(* CODESYS project SampleProject_IoDrvMasterTemplateIEC.project

Project tree, tasks and I/O mapping:
  Device : CODESYS Control Win V3, 3S - Smart Software Solutions GmbH, version 3.5.14.10
    application Application
      libraries: Standard, * (System); CAA Device Diagnosis, 3.5.15.0 (CAA Technical Workgroup)
      task MainTask (cyclic, interval t#20ms, priority 1) calls PLC_PRG
      program PLC_PRG [ST]
    My_card_IEC_Driver_master_ : My card IEC Driver (master), My company, order no. 0815, version 3.5.15.0
      Slave_without_modules_internal_8xDI_8xDO_T3 : Slave without modules (internal: 8xDI, 8xDO) T3, My company, order no. 0815, version 3.5.9.0
          settings: Slave-ID = 3
          unmapped channels: Input 8Bit, Output 8Bit
      Slave_variable_max_4_T1 : Slave variable (max 4) T1, My company, order no. 0815, version 3.5.15.0
          settings: Slave-ID = 1
        Modul_digital_input_x16_T3 : Modul digital input x16 T3, My company, order no. 0815, version 3.5.9.0
            settings: Module-ID = 3
            unmapped channels: Input 8Bit (1), Input 8Bit (2)
        Modul_digital_output_x8_T2 : Modul digital output x8 T2, My company, order no. 0815, version 3.5.9.0
            settings: Module-ID = 2
            unmapped channels: Output 8Bit, Output 8Bit
        Modul_digital_input_x8_T1 : Modul digital input x8 T1, My company, order no. 0815, version 3.5.9.0
            settings: Module-ID = 1
            unmapped channels: Input 8Bit
      Slave_variable_autoinsert_T2 : Slave variable autoinsert T2, My company, order no. 0815, version 3.5.15.0
          settings: Slave-ID = 2
        Autoinsert_1 : Modul digital input x8 T1, My company, order no. 0815, version 3.5.9.0
            settings: Module-ID = 2
            unmapped channels: Input 8Bit
        Autoinsert : Modul digital input x8 T1, My company, order no. 0815, version 3.5.9.0
            settings: Module-ID = 1
            unmapped channels: Input 8Bit
*)

// Device/Application/PLC_PRG
PROGRAM PLC_PRG
VAR

END_VAR

END_PROGRAM
